# EPICS autosave request: ipApp/Db/deviceCmdReply.req
file scalcout_settings.req P=$(P)cmdReply$(N)_formatCmd
file asynRecord.req P=$(P)cmdReply$(N)_do_IO
file scalcout_settings.req P=$(P)cmdReply$(N)_parseReply
